{attribute 'Tc2GvlVarNames'}
{attribute 'strict'}
//Tipologia Punto DiPrelievo
TYPE e_Tipo_PickPoint :
(
	RIBALTINO_NOT_DEFINED	:= -1, (* Tipologia Indefinita *)
	RIBALTINO 				:= 1, (* Ribaltino poer pacchi classico *)
	RULLIERA				:= 2, (* Rulliera Per Lastre Classica *)
	MAGAZZINO_FALDE			:= 3, (* Magazzino Falde "Statico"*)
	

	WA_CON_CASSA			:= 4, (* Postazione in di prelievo in WorkArea in CASSA *)
	WA_CON_CAVALLINA		:= 5, (* Postazione in di prelievo in WorkArea in CAVALLINA *)
	WA_CON_PALLET			:= 6  (* Postazione di prelievo in WorkArea di tipo PALLET *)
);
END_TYPE
//  RIBALTINO_NOT_DEFINED = '-1'

(* stored: Version 1.1.0.1, ProductVersion 3.1.4024.11
   EnumerationTextList e_Tipo_PickPoint: Id {b9982cb1-7328-46bf-999f-63cab6cd9646} *)
